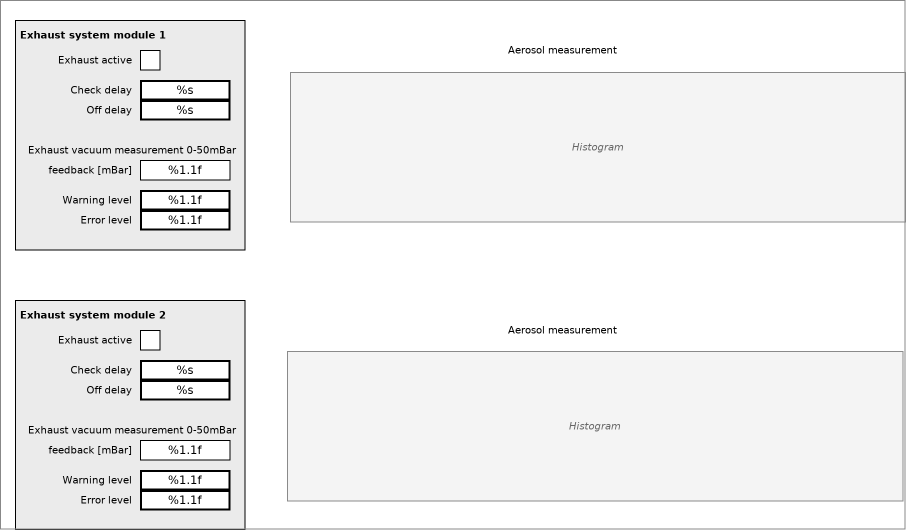
VISUALIZATION VISU_EXHAUST  // 906x530
    Rectangle (15,20 230x230)
    Rectangle (17,25 192x20), "Exhaust system module 1"
    Rectangle (45,80 90x20), "Check delay"
    Rectangle (140,80 90x20), "%s", text variable: PRG_MACHINE.fb_ExhaustSystem[1].tR_VacuumCheckDelay
        OnMouseDown: write the text variable via Edit
    Rectangle (45,100 90x20), "Off delay"
    Rectangle (140,100 90x20), "%s", text variable: PRG_MACHINE.fb_ExhaustSystem[1].tR_FUOffDelay
        OnMouseDown: write the text variable via Edit
    RoundedRectangle (140,50 20x20), colour toggle: PRG_MACHINE.fb_ExhaustSystem[1].bO_FUActivate
    Rectangle (35,50 100x20), "Exhaust active"
    Rectangle (25,140 220x20), "Exhaust vacuum measurement 0-50mBar"
    Rectangle (45,160 90x20), "feedback [mBar]"
    Rectangle (140,160 90x20), "%1.1f", text variable: PRG_MACHINE.fb_ExhaustSystem[1].fL_VacuumAnalogLevelMBar
    Histogram (290,72 616x150), scale format: %.1f, scale 0..2
        p1518820177: PRG_MACHINE.fb_ExhaustSystem[1].fL_ParticleMeasurements
        p102497268: PRG_MACHINE.fb_ExhaustSystem[1].fL_ParticleMeasurements
        p788070771: ARRAY [1..iC_ParticleMeasurementNb] OF REAL
    Rectangle (505,40 220x20), "Aerosol measurement"
    Rectangle (45,190 90x20), "Warning level"
    Rectangle (140,190 90x20), "%1.1f", text variable: PRG_MACHINE.fb_ExhaustSystem[1].fR_VacuumWarningLevelMBar
        OnMouseDown: write the text variable via Edit
    Rectangle (45,210 90x20), "Error level"
    Rectangle (140,210 90x20), "%1.1f", text variable: PRG_MACHINE.fb_ExhaustSystem[1].fR_VacuumErrorLevelMBar
        OnMouseDown: write the text variable via Edit
    Rectangle (15,300 230x230)
    Rectangle (17,305 192x20), "Exhaust system module 2"
    Rectangle (45,360 90x20), "Check delay"
    Rectangle (140,360 90x20), "%s", text variable: PRG_MACHINE.fb_ExhaustSystem[2].tR_VacuumCheckDelay
        OnMouseDown: write the text variable via Edit
    Rectangle (45,380 90x20), "Off delay"
    Rectangle (140,380 90x20), "%s", text variable: PRG_MACHINE.fb_ExhaustSystem[2].tR_FUOffDelay
        OnMouseDown: write the text variable via Edit
    RoundedRectangle (140,330 20x20), colour toggle: PRG_MACHINE.fb_ExhaustSystem[2].bO_FUActivate
    Rectangle (35,330 100x20), "Exhaust active"
    Rectangle (25,420 220x20), "Exhaust vacuum measurement 0-50mBar"
    Rectangle (45,440 90x20), "feedback [mBar]"
    Rectangle (140,440 90x20), "%1.1f", text variable: PRG_MACHINE.fb_ExhaustSystem[2].fL_VacuumAnalogLevelMBar
    Histogram (287,351 616x150), scale format: %.1f, scale 0..2
        p1518820177: PRG_MACHINE.fb_ExhaustSystem[2].fL_ParticleMeasurements
        p102497268: PRG_MACHINE.fb_ExhaustSystem[2].fL_ParticleMeasurements
        p788070771: ARRAY [1..iC_ParticleMeasurementNb] OF REAL
    Rectangle (505,320 220x20), "Aerosol measurement"
    Rectangle (45,470 90x20), "Warning level"
    Rectangle (140,470 90x20), "%1.1f", text variable: PRG_MACHINE.fb_ExhaustSystem[2].fR_VacuumWarningLevelMBar
        OnMouseDown: write the text variable via Edit
    Rectangle (45,490 90x20), "Error level"
    Rectangle (140,490 90x20), "%1.1f", text variable: PRG_MACHINE.fb_ExhaustSystem[2].fR_VacuumErrorLevelMBar
        OnMouseDown: write the text variable via Edit
END_VISUALIZATION

(* stored: Version 1.1.0.1, ProductVersion 3.1.4024.9
   Visu VISU_EXHAUST: Id {128a8423-106f-419b-b178-293a48fc0069} *)
